FUNCTION_BLOCK E_TF (* Sets the output value depending on which input event arrives. *)
  (* Standard: 61499-1-A.1; Classification: Event Processing *)
  (* Version 1.0, 2017-07-31, Marc Jakobi, HTW Berlin *)
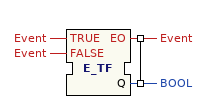
  EVENT_INPUT
    TRUE; (* Q = TRUE Event *)
    FALSE; (* Q = FALSE Event *)
  END_EVENT
  EVENT_OUTPUT
    EO WITH Q; (* Output Event *)
  END_EVENT
  VAR_OUTPUT
    Q : BOOL; (* Current Output State *)
  END_VAR
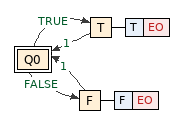
  EC_STATES
    Q0; (* Q is FALSE initially *)
    F : F -> EO; (* Reset Q and issue EO *)
    T : T -> EO; (* Set Q and issue EO *)
  END_STATES
  EC_TRANSITIONS
    Q0 TO T := TRUE;
    Q0 TO F := FALSE;
    F TO Q0 := 1;
    T TO Q0 := 1;
  END_TRANSITIONS
  ALGORITHM T IN ST: (* Set Q *)
Q:=TRUE;
  END_ALGORITHM
  ALGORITHM F IN ST: (* Reset Q *)
Q:=FALSE;
  END_ALGORITHM
END_FUNCTION_BLOCK
